// TIA Portal V20 export
DATA_BLOCK "HMI_Interface_Overview"   // DB276
// stored: Access Published, MemoryReserve 100
   VAR
      State : Struct
         "Anode Reel Cut" : "HMI_IF_OverView_Unit_UDT";
         "Cathode Reel Cut" : "HMI_IF_OverView_Unit_UDT";
         "Stacker #1" : "HMI_IF_OverView_Unit_UDT";
         "Stacker #2" : "HMI_IF_OverView_Unit_UDT";
         Inspection : "HMI_IF_OverView_Unit_UDT";
      END_STRUCT;
   END_VAR
BEGIN
   State."Anode Reel Cut".State.Communication := 0;
   State."Anode Reel Cut".State.Mode := 0;
   State."Anode Reel Cut".State.State := 0;
   State."Anode Reel Cut".State.Emergency := 0;
   State."Anode Reel Cut"."Link&Unlink".Em0 := FALSE;
   State."Anode Reel Cut"."Link&Unlink".Em1 := FALSE;
   State."Anode Reel Cut"."Link&Unlink".Em2 := FALSE;
   State."Anode Reel Cut"."Link&Unlink".Em3 := FALSE;
   State."Anode Reel Cut"."Link&Unlink".Em4 := FALSE;
   State."Anode Reel Cut"."Link&Unlink".Em5 := FALSE;
   State."Anode Reel Cut"."Link&Unlink".Em6 := FALSE;
   State."Anode Reel Cut"."Link&Unlink".Em7 := FALSE;
   State."Anode Reel Cut"."Link&Unlink".Em8 := FALSE;
   State."Anode Reel Cut"."Link&Unlink".Em9 := FALSE;
   State."Anode Reel Cut"."Link&Unlink".Em10 := FALSE;
   State."Anode Reel Cut"."Link&Unlink".Em11 := FALSE;
   State."Anode Reel Cut"."Link&Unlink".Em12 := FALSE;
   State."Anode Reel Cut"."Link&Unlink".Em13 := FALSE;
   State."Anode Reel Cut"."Link&Unlink".Em14 := FALSE;
   State."Anode Reel Cut"."Link&Unlink".Em15 := FALSE;
   State."Anode Reel Cut".Production."Total Input Quantity" := 0;
   State."Anode Reel Cut".Production."Remain Count" := 0;
   State."Anode Reel Cut".Production."Processed Count" := 0;
   State."Anode Reel Cut".Production."NG Count" := 0;
   State."Cathode Reel Cut".State.Communication := 0;
   State."Cathode Reel Cut".State.Mode := 0;
   State."Cathode Reel Cut".State.State := 0;
   State."Cathode Reel Cut".State.Emergency := 0;
   State."Cathode Reel Cut"."Link&Unlink".Em0 := FALSE;
   State."Cathode Reel Cut"."Link&Unlink".Em1 := FALSE;
   State."Cathode Reel Cut"."Link&Unlink".Em2 := FALSE;
   State."Cathode Reel Cut"."Link&Unlink".Em3 := FALSE;
   State."Cathode Reel Cut"."Link&Unlink".Em4 := FALSE;
   State."Cathode Reel Cut"."Link&Unlink".Em5 := FALSE;
   State."Cathode Reel Cut"."Link&Unlink".Em6 := FALSE;
   State."Cathode Reel Cut"."Link&Unlink".Em7 := FALSE;
   State."Cathode Reel Cut"."Link&Unlink".Em8 := FALSE;
   State."Cathode Reel Cut"."Link&Unlink".Em9 := FALSE;
   State."Cathode Reel Cut"."Link&Unlink".Em10 := FALSE;
   State."Cathode Reel Cut"."Link&Unlink".Em11 := FALSE;
   State."Cathode Reel Cut"."Link&Unlink".Em12 := FALSE;
   State."Cathode Reel Cut"."Link&Unlink".Em13 := FALSE;
   State."Cathode Reel Cut"."Link&Unlink".Em14 := FALSE;
   State."Cathode Reel Cut"."Link&Unlink".Em15 := FALSE;
   State."Cathode Reel Cut".Production."Total Input Quantity" := 0;
   State."Cathode Reel Cut".Production."Remain Count" := 0;
   State."Cathode Reel Cut".Production."Processed Count" := 0;
   State."Cathode Reel Cut".Production."NG Count" := 0;
   State."Stacker #1".State.Communication := 0;
   State."Stacker #1".State.Mode := 0;
   State."Stacker #1".State.State := 0;
   State."Stacker #1".State.Emergency := 0;
   State."Stacker #1"."Link&Unlink".Em0 := FALSE;
   State."Stacker #1"."Link&Unlink".Em1 := FALSE;
   State."Stacker #1"."Link&Unlink".Em2 := FALSE;
   State."Stacker #1"."Link&Unlink".Em3 := FALSE;
   State."Stacker #1"."Link&Unlink".Em4 := FALSE;
   State."Stacker #1"."Link&Unlink".Em5 := FALSE;
   State."Stacker #1"."Link&Unlink".Em6 := FALSE;
   State."Stacker #1"."Link&Unlink".Em7 := FALSE;
   State."Stacker #1"."Link&Unlink".Em8 := FALSE;
   State."Stacker #1"."Link&Unlink".Em9 := FALSE;
   State."Stacker #1"."Link&Unlink".Em10 := FALSE;
   State."Stacker #1"."Link&Unlink".Em11 := FALSE;
   State."Stacker #1"."Link&Unlink".Em12 := FALSE;
   State."Stacker #1"."Link&Unlink".Em13 := FALSE;
   State."Stacker #1"."Link&Unlink".Em14 := FALSE;
   State."Stacker #1"."Link&Unlink".Em15 := FALSE;
   State."Stacker #1".Production."Total Input Quantity" := 0;
   State."Stacker #1".Production."Remain Count" := 0;
   State."Stacker #1".Production."Processed Count" := 0;
   State."Stacker #1".Production."NG Count" := 0;
   State."Stacker #2".State.Communication := 0;
   State."Stacker #2".State.Mode := 0;
   State."Stacker #2".State.State := 0;
   State."Stacker #2".State.Emergency := 0;
   State."Stacker #2"."Link&Unlink".Em0 := FALSE;
   State."Stacker #2"."Link&Unlink".Em1 := FALSE;
   State."Stacker #2"."Link&Unlink".Em2 := FALSE;
   State."Stacker #2"."Link&Unlink".Em3 := FALSE;
   State."Stacker #2"."Link&Unlink".Em4 := FALSE;
   State."Stacker #2"."Link&Unlink".Em5 := FALSE;
   State."Stacker #2"."Link&Unlink".Em6 := FALSE;
   State."Stacker #2"."Link&Unlink".Em7 := FALSE;
   State."Stacker #2"."Link&Unlink".Em8 := FALSE;
   State."Stacker #2"."Link&Unlink".Em9 := FALSE;
   State."Stacker #2"."Link&Unlink".Em10 := FALSE;
   State."Stacker #2"."Link&Unlink".Em11 := FALSE;
   State."Stacker #2"."Link&Unlink".Em12 := FALSE;
   State."Stacker #2"."Link&Unlink".Em13 := FALSE;
   State."Stacker #2"."Link&Unlink".Em14 := FALSE;
   State."Stacker #2"."Link&Unlink".Em15 := FALSE;
   State."Stacker #2".Production."Total Input Quantity" := 0;
   State."Stacker #2".Production."Remain Count" := 0;
   State."Stacker #2".Production."Processed Count" := 0;
   State."Stacker #2".Production."NG Count" := 0;
   State.Inspection.State.Communication := 0;
   State.Inspection.State.Mode := 0;
   State.Inspection.State.State := 0;
   State.Inspection.State.Emergency := 0;
   State.Inspection."Link&Unlink".Em0 := FALSE;
   State.Inspection."Link&Unlink".Em1 := FALSE;
   State.Inspection."Link&Unlink".Em2 := FALSE;
   State.Inspection."Link&Unlink".Em3 := FALSE;
   State.Inspection."Link&Unlink".Em4 := FALSE;
   State.Inspection."Link&Unlink".Em5 := FALSE;
   State.Inspection."Link&Unlink".Em6 := FALSE;
   State.Inspection."Link&Unlink".Em7 := FALSE;
   State.Inspection."Link&Unlink".Em8 := FALSE;
   State.Inspection."Link&Unlink".Em9 := FALSE;
   State.Inspection."Link&Unlink".Em10 := FALSE;
   State.Inspection."Link&Unlink".Em11 := FALSE;
   State.Inspection."Link&Unlink".Em12 := FALSE;
   State.Inspection."Link&Unlink".Em13 := FALSE;
   State.Inspection."Link&Unlink".Em14 := FALSE;
   State.Inspection."Link&Unlink".Em15 := FALSE;
   State.Inspection.Production."Total Input Quantity" := 0;
   State.Inspection.Production."Remain Count" := 0;
   State.Inspection.Production."Processed Count" := 0;
   State.Inspection.Production."NG Count" := 0;
END_DATA_BLOCK
